FUNCTION_BLOCK POU IMPLEMENTS POU.controller
VAR_INPUT
END_VAR
VAR_OUTPUT
END_VAR
VAR
END_VAR

END_FUNCTION_BLOCK

(* stored: Version 1.1.0.1, ProductVersion 3.1.4024.12
   POU POU: Id {11805366-e29e-480f-a6bb-56d282f92711}, SpecialFunc None *)
